// TwinCAT 3 PLC project PLC_DemoXTS
// ProgramVersion: 3.1.4026.17
// libraries:
//   Tc2_MC2, * (Beckhoff Automation GmbH)
//   Tc2_MC2_Camming, * (Beckhoff Automation GmbH)
//   Tc2_Standard, * (Beckhoff Automation GmbH)
//   Tc2_System, * (Beckhoff Automation GmbH)
//   Tc3_Mc3Definitions, * (Beckhoff Automation GmbH)
//   Tc3_McCollisionAvoidance, * (Beckhoff Automation GmbH)
//   Tc3_McCoordinatedMotion, * (Beckhoff Automation GmbH)
//   Tc3_Module, * (Beckhoff Automation GmbH)
// project tree:
//   GVLs/ GVL_Constant.TcGVL, GVL_XTS1.TcGVL, GVL_Infeed.TcGVL
//   / PlcTask.TcTTO
//   POUs/Infeed/ FB_Infeed.TcPOU, FB_VirtualMaster.TcPOU, Prg_Camming.TcPOU
//   POUs/ MAIN.TcPOU, XTS_MAIN.TcPOU
//   POUs/XTS/ FB_MoverCheckPos.TcPOU, FB_MoverCycle.TcPOU, FB_XTS.TcPOU, FB_AllMoversToStartpos.TcPOU
//   POUs/_NEW/Mover/ FB_MoverX.TcPOU, IMover.TcIO, ST_MoverData.TcDUT
//   POUs/_NEW/Position/ FB_PositionX.TcPOU, IPosition.TcIO
//   POUs/_NEW/Station/ FB_StationX.TcPOU, IStation.TcIO
//   POUs/_NEW/TrackList/ FB_Track.TcPOU, ITrack.TcIO

CONFIGURATION PLC_DemoXTS
    RESOURCE PLC ON TwinCAT3
        TASK PlcTask(INTERVAL := T#10ms, PRIORITY := 20);
        PROGRAM MAIN WITH PlcTask : MAIN;
    END_RESOURCE
END_CONFIGURATION

// ---- POUs/_NEW/Mover/ST_MoverData.TcDUT
TYPE ST_MoverData :
STRUCT
	id : UDINT;
	pos : LREAL;
	status : INT;
	assigned : BOOL;
END_STRUCT
END_TYPE

// ---- GVLs/GVL_Constant.TcGVL
VAR_GLOBAL CONSTANT
	iMaxNumbMovers		: INT := 35;
	iMaxNumbVirtMasters	: INT := 5;
END_VAR

// ---- GVLs/GVL_XTS1.TcGVL
{attribute 'qualified_only'}
VAR_GLOBAL CONSTANT
	
	iNumbOfMovers		: INT	:= 35;
	rRailLength			: LREAL	:= 6000.0;

END_VAR


VAR_GLOBAL

	Mover				: ARRAY [1..iNumbOfMovers] OF Axis_Ref;
	CAGroup				: AXES_GROUP_REF;		

	rInitPosition		: LREAL := 1100;
	rInitVelocity		: LREAL	:= 720;
	rGap				: LREAL	:= 90;
	rMasterVelocity		: LREAL	:= 600;
	rSlaveSyncPos		: LREAL := 1300;
	rSyncDistance		: LREAL := 400;
	rXTS_Velocity		: LREAL := 720;
	rRobot1_Position	: LREAL := 4000;
	rRobot2_Position	: LREAL := 5500;
	tTime_Robot1		: TIME := T#4500MS;
	tTime_Robot2		: TIME := T#1500MS;
	
END_VAR

// ---- GVLs/GVL_Infeed.TcGVL
{attribute 'qualified_only'}
VAR_GLOBAL CONSTANT
	
	iNumbOfVirtMasters		: INT	:= 4;

END_VAR


VAR_GLOBAL

	MasterAxis				: AXIS_REF;
	VirtalMaster			: ARRAY [1..iNumbOfVirtMasters] OF Axis_Ref;

	iProductsPerMinute		: INT 	:= 60;

	rDiameterWheel			: LREAL := 480;			// Diameter Infeed Wheel
	rMasterDistance_1Cycle	: LREAL := 360;			// 8 cycles per rotation
	rSyncPosition_Wheel_XTS	: LREAL := 471.5;		
	rDetectionPosMin		: LREAL := 160;
	rDetectionPosMax		: LREAL := 200;
	
	//CamTable
	rMasterDistance_P2		: LREAL	:= 180;
	rSlaveOffset_P2			: LREAL := 0;
	rMasterDistance_P3		: LREAL	:= 20;
	rSlaveOffset_P3			: LREAL	:= 10;
	rMasterDistance_P5		: LREAL := 30;
	rSlaveOffset_P5			: LREAL;
	rMasterDistance_P6		: LREAL := 180;
	rSlaveOffset_P6			: LREAL := -5;
	rSlaveOffset			: LREAL;
	
END_VAR

// ---- POUs/_NEW/Mover/IMover.TcIO
INTERFACE IMover

METHOD AssignAxisRef : bool
VAR_INPUT
	axis : REFERENCE TO AXIS_REF;
END_VAR
END_METHOD

METHOD AssignID : bool
VAR_INPUT
	ID : UDINT;
END_VAR
END_METHOD

METHOD GetPosition : LREAL
VAR_INPUT
END_VAR
END_METHOD

METHOD GetStatus : int
VAR_INPUT
END_VAR
END_METHOD

METHOD SetPositionID : BOOL
VAR_INPUT
	ID: UDINT;
END_VAR
END_METHOD

METHOD SetStatus : BOOL;
VAR_INPUT
	status : INT;
END_VAR
END_METHOD

METHOD UpdateData : ST_MoverData
VAR_INPUT
END_VAR
END_METHOD

METHOD UpdatePosition : bool
VAR_INPUT
END_VAR
END_METHOD

END_INTERFACE

// ---- POUs/_NEW/Position/IPosition.TcIO
INTERFACE IPosition

METHOD Available : bool
VAR_INPUT
END_VAR
END_METHOD

METHOD Disable : BOOL
VAR_INPUT
END_VAR
END_METHOD

METHOD Enable : BOOL
VAR_INPUT
END_VAR
END_METHOD

METHOD GetID : UDINT
VAR_INPUT
END_VAR
END_METHOD

METHOD GetPosition : LREAL
VAR_INPUT
END_VAR
END_METHOD

METHOD SetID : BOOL
VAR_INPUT
	ID : UDINT;
END_VAR
END_METHOD

METHOD SetMover : bool
VAR_INPUT
	moverNumber : UDINT;
END_VAR
END_METHOD

METHOD SetPosition
VAR_INPUT
	position : LREAL;
END_VAR
END_METHOD

END_INTERFACE

// ---- POUs/_NEW/Station/IStation.TcIO
INTERFACE IStation

METHOD FindMoverMatch : udint
VAR_INPUT
END_VAR
END_METHOD

METHOD FindNextPosition : IPosition;
VAR_INPUT
END_VAR
END_METHOD

METHOD GetMovers : BOOL
VAR_INPUT
END_VAR
END_METHOD

METHOD SetPosRef : BOOL
VAR_INPUT
	PosIndex : DINT;
	PosRef	: REFERENCE TO FB_PositionX;
END_VAR
END_METHOD

METHOD SetStationAttraction : BOOL
VAR_INPUT
	setState : INT;
END_VAR
END_METHOD

METHOD SetTrackRef : BOOL
VAR_INPUT
	TrackRef : ITrack;
END_VAR
END_METHOD

END_INTERFACE

// ---- POUs/_NEW/TrackList/ITrack.TcIO
INTERFACE ITrack

METHOD FindMover : UDINT
VAR_INPUT
	status : INT;
END_VAR
END_METHOD

METHOD SetMoverInUse : BOOL;
VAR_INPUT
	moverNumber	: UDINT;
END_VAR
END_METHOD

METHOD SetMoverRef : BOOL
VAR_INPUT
	index : DINT;
	mover	: IMover;
END_VAR
END_METHOD

METHOD Sort : bool
VAR_INPUT
END_VAR
END_METHOD

METHOD UpdateMoverData : bool
VAR_INPUT
	data	: ST_MoverData;
END_VAR
END_METHOD

END_INTERFACE

// ---- POUs/MAIN.TcPOU
PROGRAM MAIN
VAR

	bEnable_XTS1			: BOOL;
	bMoveToStartPos_XTS1	: BOOL;
	bEnable_Master			: BOOL;
	bMoveMaster				: BOOL;
	bSensor_Product			: BOOL;

	fbInfeed1				: FB_Infeed;
	fbXTS1					: FB_XTS;
	fbMoveToStartPos_XTS1	: FB_AllMoversToStartpos;
	
	// Cycle
	i,j						: INT;
	bStartSyncMaster		: BOOL;
	bStartSyncMover			: BOOL;
	Trg_bStartSyncMaster	: R_Trig;
	iMoverAtStartpos_XTS1	: INT;
	iVirtMasterAtStartpos	: INT;
	fbMoveratStartPos_XTS1	: ARRAY [1..GVL_XTS1.iNumbOfMovers] OF FB_MoverCheckPos;
	fbMoveratRobot1Pos		: ARRAY [1..GVL_XTS1.iNumbOfMovers] OF FB_MoverCheckPos;
	fbMoveratRobot2Pos		: ARRAY [1..GVL_XTS1.iNumbOfMovers] OF FB_MoverCheckPos;
	fbMoverCycle_XTS1		: ARRAY [1..GVL_XTS1.iNumbOfMovers] OF FB_MoverCycle;
	
	// Robot1 and Robot2
	MoverAtRobot1			: ARRAY [1..10] OF INT;
	MoverAtRobot2			: ARRAY [1..10] OF INT;
	bRobot1_Filled			: BOOL;
	bRobot2_Filled			: BOOL;
	fbRobot1_Timer			: TON;
	fbRobot2_Timer			: TON;
	
	MyXTS	: XTS_MAIN;

END_VAR

Prg_Camming();

// Infeed
fbInfeed1(
	bEnable_Master		:= bEnable_Master, 
	bMoveMaster			:= bMoveMaster, 
	bSensorProduct		:= bSensor_Product,
	Master				:= GVL_Infeed.MasterAxis, 
	VirtMaster			:= GVL_Infeed.VirtalMaster,
	);


// XTS 1 : Enable all movers with Collision Avoindance
fbXTS1(
	bEnable_XTS		:= bEnable_XTS1, 
	Mover			:= GVL_XTS1.Mover, 
	CAGroup			:= GVL_XTS1.CAGroup, 
	);
	
	
// XTS 1 : Move all movers to Startposition 
fbMoveToStartPos_XTS1(
	bXTS_MoveToStartPos	:= bMoveToStartPos_XTS1, 
	rInitPosition		:= GVL_XTS1.rInitPosition, 
	rInitVelocity		:= GVL_XTS1.rInitVelocity, 
	rRailLength			:= GVL_XTS1.rRailLength, 
	rGap				:= GVL_XTS1.rGap, 
	Mover				:= GVL_XTS1.Mover,
	);

	
// XTS 1 : Find which mover is waiting at Startposition	
iMoverAtStartpos_XTS1 := 0;
FOR i:=1 TO GVL_XTS1.iNumbOfMovers DO
	fbMoveratStartPos_XTS1[i](
		rActualPosition	:= GVL_XTS1.Mover[i].NcToPlc.ModuloSetPos, 
		rCheckPosition	:= GVL_XTS1.rInitPosition, 
		rRailLength		:= GVL_XTS1.rRailLength
		);
	IF fbMoveratStartPos_XTS1[i].bInPosition THEN
		iMoverAtStartpos_XTS1 := i;
	END_IF
	
END_FOR
	
// Start Synchronisation Virtual Master
bStartSyncMaster:=FALSE;
iVirtMasterAtStartpos:=0;
FOR i := 1 TO GVL_Infeed.iNumbOfVirtMasters DO
	IF (GVL_Infeed.VirtalMaster[i].NcToPlc.SetPos>GVL_Infeed.rSlaveOffset+10) AND (GVL_Infeed.VirtalMaster[i].NcToPlc.SetPos<GVL_Infeed.rSlaveOffset+120) THEN
		iVirtMasterAtStartpos:=i;
		bStartSyncMaster:=TRUE;
	END_IF
END_FOR

// Start Synchronisation Mover
Trg_bStartSyncMaster(Clk:=bStartSyncMaster);
IF (iMoverAtStartpos_XTS1<>0) AND Trg_bStartSyncMaster.Q THEN
	bStartSyncMover:=TRUE;
END_IF
IF iMoverAtStartpos_XTS1=0 OR NOT bStartSyncMaster THEN
	bStartSyncMover:=FALSE;
END_IF

// XTS 1 : Cyclic movement for all movers
FOR i:=1 TO GVL_XTS1.iNumbOfMovers DO
	fbMoverCycle_XTS1[i](
		bStartCycle			:= bStartSyncMover AND (iMoverAtStartpos_XTS1=i), 
		iVirtMasterAtStart	:= iVirtMasterAtStartpos,
		rMasterSyncPos		:= 300,
		rSlaveSyncPos		:= (GVL_XTS1.Mover[i].NcToPlc.ModuloActTurns * GVL_XTS1.rRailLength) + GVL_XTS1.rSlaveSyncPos,
		Mover				:= GVL_XTS1.Mover[i]
		);

END_FOR

// Cyclus Pers + Robot1 

FOR j := 1 TO 10 DO
	MoverAtRobot1[j] := 0;
	FOR i:=1 TO GVL_XTS1.iNumbOfMovers DO
		fbMoveratRobot1Pos[i](
			rActualPosition	:= GVL_XTS1.Mover[i].NcToPlc.ModuloSetPos, 
			rCheckPosition	:= GVL_XTS1.rRobot1_Position - (j*GVL_XTS1.rGap) + GVL_XTS1.rGap , 
			rRailLength		:= GVL_XTS1.rRailLength
			);
		IF fbMoveratRobot1Pos[i].bInPosition THEN
			MoverAtRobot1[j] := i;
		END_IF
	END_FOR
END_FOR

bRobot1_Filled := TRUE;
FOR i := 1 TO 10 DO
	IF MoverAtRobot1[i]=0 THEN
		bRobot1_Filled := FALSE;
	END_IF
END_FOR

fbRobot1_Timer(IN:=bRobot1_Filled , PT:=GVL_XTS1.tTime_Robot1 );
IF fbRobot1_Timer.Q THEN
	FOR i:=1 TO 10 DO
		fbMoverCycle_XTS1[MoverAtRobot1[i]].Robot1_Ready:=TRUE;	
	END_FOR
ELSE
	FOR i:=1 TO GVL_XTS1.iNumbOfMovers DO
		fbMoverCycle_XTS1[i].Robot1_Ready:=FALSE;	
	END_FOR	
END_IF


// Cyclus Robot2 

FOR j := 1 TO 10 DO
	MoverAtRobot2[j] := 0;
	FOR i:=1 TO GVL_XTS1.iNumbOfMovers DO
		fbMoveratRobot2Pos[i](
			rActualPosition	:= GVL_XTS1.Mover[i].NcToPlc.ModuloSetPos, 
			rCheckPosition	:= GVL_XTS1.rRobot2_Position - (j*GVL_XTS1.rGap) + GVL_XTS1.rGap , 
			rRailLength		:= GVL_XTS1.rRailLength
			);
		IF fbMoveratRobot2Pos[i].bInPosition THEN
			MoverAtRobot2[j] := i;
		END_IF
	END_FOR
END_FOR

bRobot2_Filled := TRUE;
FOR i := 1 TO 10 DO
	IF MoverAtRobot2[i]=0 THEN
		bRobot2_Filled := FALSE;
	END_IF
END_FOR

fbRobot2_Timer(IN:=bRobot2_Filled , PT:=GVL_XTS1.tTime_Robot2 );
IF fbRobot2_Timer.Q THEN
	FOR i:=1 TO 10 DO
		fbMoverCycle_XTS1[MoverAtRobot2[i]].Robot2_Ready:=TRUE;	
	END_FOR
ELSE
	FOR i:=1 TO GVL_XTS1.iNumbOfMovers DO
		fbMoverCycle_XTS1[i].Robot2_Ready:=FALSE;	
	END_FOR	
END_IF

// call
MyXTS(axisRef := GVL_XTS1.Mover);

END_PROGRAM

// ---- POUs/Infeed/FB_Infeed.TcPOU
FUNCTION_BLOCK FB_Infeed
VAR_INPUT
	bEnable_Master			: BOOL;
	bMoveMaster				: BOOL;
	bSensorProduct			: BOOL;
END_VAR

VAR_IN_OUT
	Master					: Axis_Ref;
	VirtMaster				: ARRAY [*] OF Axis_Ref;
END_VAR

VAR
	i						: DINT;
	iStartIndex				: DINT;
	VeloMaster				: LREAL;
	bToggle					: BOOL;

	fbPowerMaster			: MC_Power;
	fbMoveMaster			: MC_MoveVelocity;
	fbStopMaster			: MC_Halt;
	fbPowerVirtMaster		: ARRAY [1..iMaxNumbVirtMasters] OF MC_Power;
	fbVirtMaster			: ARRAY [1..iMaxNumbVirtMasters] OF FB_VirtualMaster;

END_VAR

// Enable Master
Master.ReadStatus();
fbPowerMaster(
	Axis			:= Master, 
	Enable			:= bEnable_Master, 
	Enable_Positive	:= bEnable_Master, 
	Enable_Negative	:= bEnable_Master, 
	Override		:= 100, 
	);
	
FOR i := 1 TO UPPER_BOUND(VirtMaster,1) DO
	VirtMaster[i].ReadStatus();
	fbPowerVirtMaster[i](
		Axis			:= VirtMaster[i], 
		Enable			:= bEnable_Master, 
		Enable_Positive	:= bEnable_Master, 
		Enable_Negative	:= bEnable_Master, 
		Override		:= 100, 
		);
END_FOR


// Start-Stop Master

VeloMaster := GVL_Infeed.iProductsPerMinute * 360 / 60;
bToggle:=NOT bToggle;

fbMoveMaster(
	Axis		:= Master, 
	Execute		:= bMoveMaster AND bToggle, 
	Velocity	:= VeloMaster, 
	Direction	:= MC_Positive_Direction, 
	);
fbStopMaster(
	Axis		:= Master, 
	Execute		:= NOT bMoveMaster, 
	);

// Virtual Master ready to start
iStartIndex:=0;
FOR i := 1 TO UPPER_BOUND(VirtMaster,1) DO
	IF VirtMaster[i].NcToPlc.ActPos=0 THEN
		iStartIndex:=i;
		i:=5;
	END_IF
END_FOR
	
// Detection product
FOR i := 1 TO UPPER_BOUND(VirtMaster,1) DO
	fbVirtMaster[i].bActivateCam:=FALSE;
END_FOR

IF (Master.NcToPlc.ModuloActPos > GVL_Infeed.rDetectionPosMin) AND (Master.NcToPlc.ModuloActPos < GVL_Infeed.rDetectionPosMax) AND bSensorProduct THEN
	fbVirtMaster[iStartIndex].bActivateCam:=TRUE;
END_IF
 
FOR i := 1 TO UPPER_BOUND(VirtMaster,1) DO
	fbVirtMaster[i](
		Master:= Master, 
		Slave:= VirtMaster[i],
		);
END_FOR

END_FUNCTION_BLOCK

// ---- POUs/Infeed/FB_VirtualMaster.TcPOU
FUNCTION_BLOCK FB_VirtualMaster
VAR_INPUT
	bActivateCam	: BOOL;
END_VAR
VAR_OUTPUT
END_VAR
VAR_IN_OUT
	Master			: Axis_Ref;
	Slave			: Axis_Ref;
END_VAR
VAR
	fbCamIn			: MC_CamIn;
	Options			: ST_CamInOptions;
	fbCamOut		: MC_CamOut;
	fbStop			: MC_Halt;
	fbSetPos		: MC_SetPosition;
	MasterOffset	: LREAL;;
END_VAR

Options.ActivationMode := MC_CamActivationMode.MC_CAMACTIVATION_ATMASTERAXISPOS;
Options.ActivationPosition := (Master.NcToPlc.ModuloActTurns+1)*360;
CASE (Master.NcToPlc.ModuloActTurns MOD 3) OF
0:	MasterOffset:=720;
1:	MasterOffset:=360;
2:	MasterOffset:=0;
END_CASE


fbCamIn(
	Master			:= Master, 
	Slave			:= Slave, 
	Execute			:= bActivateCam, 
	StartMode		:= MC_StartMode.MC_STARTMODE_MASTERABS_SLAVEREL,
	MasterOffset	:= MasterOffset,
	CamTableID		:= 1, 
	Options			:= Options, 
	);

fbCamOut.Execute	:= FALSE;
fbStop.Execute 		:= FALSE;
fbSetPos.Execute 	:= FALSE;
IF Slave.NcToPlc.ActPos>750 THEN
	fbCamOut.Execute := TRUE;
	IF fbCamOut.Done THEN fbStop.Execute := TRUE; END_IF
	IF fbStop.Done THEN fbSetPos.Execute := TRUE; END_IF
END_IF

fbCamOut	(Slave	:= Slave);	
fbStop		(Axis	:= Slave);
fbSetPos	(Axis	:= Slave);

END_FUNCTION_BLOCK

// ---- POUs/XTS/FB_XTS.TcPOU
FUNCTION_BLOCK FB_XTS

VAR_INPUT
	bEnable_XTS				: BOOL;
END_VAR

VAR_IN_OUT
	Mover					: ARRAY [*] OF AXIS_REF;
	CAGroup					: AXES_GROUP_REF;
END_VAR

VAR_OUTPUT
	// Status bits	
	bAllMoversFound			: BOOL;
	bAllMoversEnabled		: BOOL;
	bMoverHasError			: BOOL;
	bCAGroupMoving			: BOOL;
	bCAGroupError			: BOOL;
	bCAGroupNotReady		: BOOL;
	bCAGroupStandby			: BOOL;
	bCAGroupStopping		: BOOL;
	bCAGroupDisabled		: BOOL;
END_VAR

VAR
	i						: DINT;
	step					: INT;
	pMover					: POINTER TO AXIS_REF;

	// Command bits
	bResetAll				: BOOL;
	bEnableAllMovers		: BOOL;
	bEnableCAGroup			: BOOL;
	bDisableCAGroup			: BOOL;
	bResetMovers			: BOOL;
	bResetCAGroup			: BOOL;
	bConfig_CAGroup			: BOOL;
	bReConfig_CAGroup		: BOOL;

	// Status bits	
	bRunXTS					: BOOL;
	bConfig_CAGroupDone		: BOOL;
	bConfig_CAGroupErr		: BOOL;
	bReConfig_CAGroupDone	: BOOL;
	bReConfig_CAGroupErr	: BOOL;

	// Function Blocks
	fbPowerMover			: ARRAY [1..iMaxNumbMovers] OF MC_Power;
	fbResetMover			: ARRAY [1..iMaxNumbMovers] OF MC_Reset;
	fbAddAxisTo_CAGroup		: ARRAY [1..iMaxNumbMovers] OF MC_AddAxisToGroup;
	fbRemoveFrom_CAGroup	: ARRAY [1..iMaxNumbMovers] OF MC_RemoveAxisFromGroup;
	fbEnableCAGroup			: MC_GroupEnable;
	fbDisableCAGroup		: MC_GroupDisable;
	fbResetCAGroup			: MC_GroupReset;
	fbCAGroupReadStatus		: MC_GroupReadStatus;
	fbTimer					: TON;
	fbRTrgReset				: R_TRIG;	
END_VAR


// **************************************************************************************
// Wait until XTS is started
// **************************************************************************************

IF NOT bRunXTS THEN
	bAllMoversFound := TRUE;
	FOR i:=1 TO UPPER_BOUND(Mover,1) DO
		bAllMoversFound := bAllMoversFound AND Mover[i].NcToPlc.ActPos<>0;
	END_FOR
	bRunXTS := bAllMoversFound;
END_IF

IF NOT bRunXTS THEN
	RETURN;
END_IF


// **************************************************************************************
// Init XTS with Collision Avoidance
// **************************************************************************************

CASE step OF
	
0:		// Wait for Enable-XTS command
		bResetCAGroup 			:= fbRTrgReset.Q;
		bResetMovers			:= fbRTrgReset.Q;	 
		bEnableCAGroup			:= FALSE;
		bDisableCAGroup			:= FALSE;
		bConfig_CAGroupDone		:= FALSE;
		bConfig_CAGroupErr		:= FALSE;
		bReConfig_CAGroupDone	:= FALSE;
		bReConfig_CAGroupErr	:= FALSE;
		IF bEnable_XTS THEN
			Step:=10;	
		END_IF
	
10:		//Add Axis to Group
		bConfig_CAGroup:=TRUE;
		IF bConfig_CAGroupDone THEN
			Step:=20;
			bConfig_CAGroup:=FALSE;
		END_IF
		IF bConfig_CAGroupErr THEN
			Step:=999;
			bConfig_CAGroup:=FALSE;
		END_IF
		
20:		//Enable CA-Group
		bEnableCAGroup:=TRUE;
		IF fbEnableCAGroup.Done THEN
			Step:=30;
			bEnableCAGroup:=FALSE;
		END_IF
		IF fbEnableCAGroup.Error THEN
			Step:=999;
			bEnableCAGroup:=FALSE;
		END_IF	
		
30:		// Power Movers
		bEnableAllMovers := TRUE;
		fbTimer(IN:=TRUE,PT:=T#200MS);
		IF fbTimer.Q THEN
			Step:=40;
			fbTimer(IN:=FALSE);
		END_IF
			
40:		// Reset Movers
		bResetMovers := TRUE;
		fbTimer(IN:=TRUE,PT:=T#2000MS);
		IF bAllMoversEnabled THEN
			Step:=50;
			bResetMovers := FALSE;
			fbTimer(IN:=FALSE);
		END_IF
		IF fbTimer.Q THEN 
			Step:=999;
			bResetMovers := FALSE;
			fbTimer(IN:=FALSE);
		END_IF
	
50:		// Reset CA-Group
		bResetCAGroup := TRUE;
		IF fbResetCAGroup.Done THEN
			Step:=100;
			bResetCAGroup := FALSE;
		END_IF
		IF fbResetCAGroup.Error THEN
			Step:=999;
			bResetCAGroup := FALSE;
		END_IF	
	
100:	// XTS CA-Group Ready
		bResetCAGroup 	:= fbRTrgReset.Q;
		bResetMovers	:= fbRTrgReset.Q;	 
		IF NOT bEnable_XTS THEN
			Step:=110;
		END_IF

110:	// Disable Movers
		bEnableAllMovers := FALSE;
		fbTimer(IN:=TRUE,PT:=T#200MS);
		IF fbTimer.Q THEN
			Step:=120;
			fbTimer(IN:=FALSE);
		END_IF
	
120:	// Disable CA-Group		
		bDisableCAGroup:=TRUE;
		IF fbDisableCAGroup.Done THEN
			Step:=130;
			bDisableCAGroup:=FALSE;
			bEnableAllMovers:=FALSE;
		END_IF
		IF fbDisableCAGroup.Error THEN
			Step:=999;
			bDisableCAGroup:=FALSE;
		END_IF		

130:	// Reconfig CA-Group
		bReConfig_CAGroup:=TRUE;
		IF bReConfig_CAGroupDone THEN
			Step:=140;
			bReConfig_CAGroup:=FALSE;
		END_IF
		IF bReConfig_CAGroupErr THEN
			Step:=999;
			bReConfig_CAGroup:=FALSE;
		END_IF
		M_Config_CAGroup();
		
140:	// Reset Movers
		bResetMovers := TRUE;
		fbTimer(IN:=TRUE,PT:=T#2000MS);
		IF NOT bMoverHasError THEN
			Step:=150;
			bResetMovers := FALSE;
			fbTimer(IN:=FALSE);
		END_IF
		IF fbTimer.Q THEN 
			Step:=999;
			bResetMovers := FALSE;
			fbTimer(IN:=FALSE);
		END_IF

150:	// Reset CA-Group
		bResetCAGroup := TRUE;
		IF fbResetCAGroup.Done THEN
			Step:=0;
			bResetCAGroup := FALSE;
		END_IF
		IF fbResetCAGroup.Error THEN
			Step:=999;
			bResetCAGroup := FALSE;
		END_IF	

999:	// Error
		bEnable_XTS			:=FALSE;
		bEnableAllMovers	:=FALSE;
		bResetCAGroup 		:= fbRTrgReset.Q;
		bResetMovers		:= fbRTrgReset.Q;	 
		IF fbRTrgReset.Q THEN
			Step:=0;
		END_IF

END_CASE

M_Config_CAGroup();
M_ReadStatus();
M_Enable_Movers();
M_Enable_CAGroup();
M_Reset();	

fbRTrgReset(CLK:=bResetAll);

METHOD M_Config_CAGroup 	: BOOL
VAR
END_VAR
// Add Axis to Group
FOR i := 1 TO UPPER_BOUND(Mover,1) DO
	bConfig_CAGroupDone	:= TRUE;
	fbAddAxisTo_CAGroup[i](
		AxesGroup		:= CAGroup, 
		Axis			:= Mover[i], 
		Execute			:= bConfig_CAGroup, 
		IdentInGroup	:= UDINT_TO_IDENTINGROUP(i), 
		);		
	bConfig_CAGroupDone	:= bConfig_CAGroupDone AND fbAddAxisTo_CAGroup[i].Done;
	bConfig_CAGroupErr	:= bConfig_CAGroupErr OR fbAddAxisTo_CAGroup[i].Error;
END_FOR

// Remove Axis from Group
FOR i := 1 TO UPPER_BOUND(Mover,1) DO
	bReConfig_CAGroupDone	:= TRUE;
	fbRemoveFrom_CAGroup[i](
		AxesGroup			:= CAGroup, 
		Execute				:= bReConfig_CAGroup, 
		IdentInGroup		:= UDINT_TO_IDENTINGROUP(i), 
		);
	bReConfig_CAGroupDone	:= bReConfig_CAGroupDone AND fbRemoveFrom_CAGroup[i].Done;
	bReConfig_CAGroupErr	:= bReConfig_CAGroupErr OR fbRemoveFrom_CAGroup[i].Error;
END_FOR
END_METHOD

METHOD M_Enable_CAGroup : BOOL
VAR_INPUT
END_VAR
// Enable CA-Group
fbEnableCAGroup(
	AxesGroup	:= CAGroup, 
	Execute		:= bEnableCAGroup, 
	);	

	
// Disable CA-Group	
fbDisableCAGroup(
	AxesGroup	:= CAGroup, 
	Execute		:= bDisableCAGroup, 
	);
END_METHOD

METHOD M_Enable_Movers : BOOL
VAR_INPUT
END_VAR
// Enable Movers
FOR i:=1 TO UPPER_BOUND(Mover,1) DO
	fbPowerMover[i](
		Axis			:= Mover[i], 
		Enable			:= bEnableAllMovers, 
		Enable_Positive	:= bEnableAllMovers, 
		Enable_Negative	:= bEnableAllMovers, 
		Override		:= 100, 
		);
END_FOR
END_METHOD

METHOD M_ReadStatus : BOOL
VAR_INPUT
END_VAR
// All Movers Enabled
bAllMoversEnabled := TRUE;
FOR i:=1 TO UPPER_BOUND(Mover,1) DO
	bAllMoversEnabled := bAllMoversEnabled AND Mover[i].Status.ControlLoopClosed;
END_FOR

// Mover has Error
bMoverHasError := FALSE;
FOR i:=1 TO UPPER_BOUND(Mover,1) DO
	bMoverHasError := bMoverHasError OR Mover[i].Status.Error;
END_FOR

// Read Status NC
FOR i:=1 TO UPPER_BOUND(Mover,1) DO
	Mover[i].ReadStatus();
END_FOR

// Read Status CA-Group
fbCAGroupReadStatus(
	AxesGroup		:= CAGroup, 
	Enable			:= NOT fbCAGroupReadStatus.Busy, 
	GroupMoving		=> bCAGroupMoving, 
	GroupErrorStop	=> bCAGroupError, 
	GroupNotReady	=> bCAGroupNotReady, 
	GroupStandby	=> bCAGroupStandby, 
	GroupStopping	=> bCAGroupStopping, 
	GroupDisabled	=> bCAGroupDisabled, 
	);
END_METHOD

METHOD M_Reset : BOOL
VAR_INPUT
END_VAR
// Reset Movers
FOR i:=1 TO UPPER_BOUND(Mover,1) DO
	fbResetMover[i](
		Axis	:= Mover[i], 
		Execute	:= bResetMovers (*AND Mover[i].Status.Error*) 
		);
END_FOR

// Reset CA-Group
fbResetCAGroup(
	AxesGroup	:= CAGroup, 
	Execute		:= bResetCAGroup, 
	);
END_METHOD

END_FUNCTION_BLOCK

// ---- POUs/XTS/FB_AllMoversToStartpos.TcPOU
FUNCTION_BLOCK FB_AllMoversToStartpos
VAR_INPUT
	bXTS_MoveToStartPos		: BOOL;
	rInitPosition			: LREAL;
	rInitVelocity			: LREAL;
	rRailLength				: LREAL;
	rGap					: LREAL;
END_VAR

VAR_IN_OUT
	Mover					: ARRAY [*] OF AXIS_REF;
END_VAR

VAR
	i						: DINT;
	fbMoveToStartPos		: ARRAY [1..iMaxNumbMovers] OF MC_MoveRelativeCA;
END_VAR

// **************************************************************************************
// Move all Movers to initial position
// **************************************************************************************

FOR i:=1 TO UPPER_BOUND(Mover,1) DO
	
	IF Mover[i].NcToPlc.ModuloSetPos < (rInitPosition - 1) THEN
		fbMoveToStartPos[i].Distance := rInitPosition - Mover[i].NcToPlc.ModuloSetPos;
	ELSE;
		fbMoveToStartPos[i].Distance := rInitPosition - Mover[i].NcToPlc.ModuloSetPos + rRailLength ;
	END_IF
		
	fbMoveToStartPos[i](
		Axis			:= Mover[i], 
		Execute			:= bXTS_MoveToStartPos, 
		ContinuousUpdate:= TRUE, 
		Velocity		:= rInitVelocity, 
		Gap				:= rGap, 
		);

END_FOR

END_FUNCTION_BLOCK

// ---- POUs/XTS/FB_MoverCheckPos.TcPOU
FUNCTION_BLOCK FB_MoverCheckPos
VAR_INPUT
	rActualPosition	: LREAL;
	rCheckPosition	: LREAL;
	rRailLength		: LREAL;
END_VAR
VAR_OUTPUT
	bInPosition		: BOOL;
END_VAR
VAR
	rTolerance		: LREAL	:= 1;
END_VAR

bInPosition:=FALSE;
IF rCheckPosition<=rTolerance THEN
	IF rActualPosition>(rRailLength+rCheckPosition-rTolerance) OR rActualPosition<(rCheckPosition+rTolerance) THEN
		bInPosition:=TRUE;
	END_IF
END_IF

IF rCheckPosition>rTolerance AND rCheckPosition<(rRailLength-rTolerance) THEN
	IF rActualPosition>(rCheckPosition-rTolerance) AND rActualPosition<(rCheckPosition+rTolerance)THEN
		bInPosition:=TRUE;
	END_IF
END_IF

IF rCheckPosition>=(rRailLength-rTolerance) THEN
	IF rActualPosition>(rCheckPosition-rTolerance) OR rActualPosition<(rCheckPosition+rTolerance-rRailLength)THEN
		bInPosition:=TRUE;
	END_IF
END_IF

END_FUNCTION_BLOCK

// ---- POUs/XTS/FB_MoverCycle.TcPOU
FUNCTION_BLOCK FB_MoverCycle 
VAR_INPUT
	bStartCycle			: BOOL;
	iVirtMasterAtStart	: int;
	rMasterSyncPos		: MC_LREAL;
	rSlaveSyncPos		: MC_LREAL;
	Robot1_Ready		: BOOL;
	Robot2_Ready		: BOOL;
END_VAR
VAR_OUTPUT
END_VAR
VAR_IN_OUT
	Mover				: AXIS_REF;
END_VAR
VAR
	i					: INT;
	step				: INT;
	fbGearIn			: MC_GearInPosCA;
	fbMoveToRobot1		: MC_MoveAbsoluteCA;
	fbMoveToRobot2		: MC_MoveAbsoluteCA;
	fbMoveStartPos		: MC_MoveAbsoluteCA;
END_VAR

CASE step OF
	
	0:	// Wait for startcommand
	
		fbGearIn.Execute		:= FALSE;	
		fbMoveStartPos.Execute 	:= FALSE;
		fbMoveToRobot1.Execute	:= FALSE;	
		fbMoveToRobot2.Execute	:= FALSE;	
	
		IF bStartCycle THEN
			step:=10;
		END_IF
		
	
	10:	// Sync with Master

		fbGearIn.Execute				:= TRUE; 
		fbGearIn.ContinuousUpdate		:= TRUE; 
		fbGearIn.RatioNumerator			:= 1; 
		fbGearIn.RatioDenumerator		:= 1; 
		fbGearIn.MasterSyncPosition		:= rMasterSyncPos; 
		fbGearIn.SlaveSyncPosition		:= rSlaveSyncPos; 
		fbGearIn.SyncStrategy			:= mcSyncStrategyEarly; 
		fbGearIn.Velocity				:= 4000;

		IF Mover.NcToPlc.ModuloActPos > (GVL_XTS1.rSlaveSyncPos+GVL_XTS1.rSyncDistance) THEN
			step:=20;
		END_IF

	20:	// Move To Robot1	
		
		fbMoveToRobot1.Position			:= (Mover.NcToPlc.ModuloActTurns * GVL_XTS1.rRailLength) + GVL_XTS1.rRobot1_Position;
		fbMoveToRobot1.Velocity 		:= GVL_XTS1.rXTS_Velocity;
		fbMoveToRobot1.ContinuousUpdate	:= FALSE;
		fbMoveToRobot1.Gap				:= GVL_XTS1.rGap;
		fbMoveToRobot1.BufferMode		:= mcAborting;
		fbMoveToRobot1.Execute			:= TRUE;
		
		IF Robot1_Ready THEN
			step:=30;
		END_IF
		
	30:	// Move To Robot2	
		
		fbMoveToRobot2.Position			:= (Mover.NcToPlc.ModuloActTurns * GVL_XTS1.rRailLength) + GVL_XTS1.rRobot2_Position;
		fbMoveToRobot2.Velocity 		:= GVL_XTS1.rXTS_Velocity;
		fbMoveToRobot2.ContinuousUpdate	:= FALSE;
		fbMoveToRobot2.Gap				:= GVL_XTS1.rGap;
		fbMoveToRobot2.BufferMode		:= mcAborting;
		fbMoveToRobot2.Execute			:= TRUE;
		
		IF Robot2_Ready THEN
			step:=40;
		END_IF
	
	40:	// Goto startposition

		fbMoveStartPos.Position			:= (Mover.NcToPlc.ModuloActTurns * GVL_XTS1.rRailLength) + GVL_XTS1.rInitPosition + GVL_XTS1.rRailLength;
		fbMoveStartPos.Velocity 		:= GVL_XTS1.rXTS_Velocity;
		fbMoveStartPos.ContinuousUpdate	:= FALSE;
		fbMoveStartPos.Gap				:= GVL_XTS1.rGap;
		fbMoveStartPos.BufferMode		:= mcAborting;
		fbMoveStartPos.Execute			:= TRUE;
		IF fbMoveStartPos.Done THEN
			step:=0;
		END_IF
		

END_CASE

fbMoveStartPos	( Axis:= Mover);
fbMoveToRobot1	( Axis:= Mover);
fbMoveToRobot2	( Axis:= Mover);
fbGearIn		( Master:= GVL_Infeed.VirtalMaster[iVirtMasterAtStart], Slave:= Mover);

END_FUNCTION_BLOCK

// ---- POUs/XTS_MAIN.TcPOU
FUNCTION_BLOCK XTS_MAIN
VAR_IN_OUT
	axisRef : ARRAY [1..iMaxNumbMovers] OF AXIS_REF;
END_VAR
VAR
	fbMover	: ARRAY [1..iMaxNumbMovers] OF FB_MoverX;
	fbPosition	: ARRAY [1..10] OF FB_PositionX;
	initDone : BOOL;
	i : DINT;
	positionActive : DINT;
	size : DINT;
	position : INT;
	list : ARRAY [1..iMaxNumbMovers] OF ST_MoverData;
	trackList : FB_Track;
	foundMover : UDINT;
	id : UDINT;
	IPosition : IPosition;
	IMover : IMover;
	statusRequest : INT := 1;
	station : FB_StationX;

END_VAR

// Init
IF NOT initDone THEN
	// Reference Axis to Mover Object
	FOR i:=1 TO iMaxNumbMovers DO
		fbMover[i].AssignID(ID:= i);
		fbMover[i].AssignAxisRef(axis:= axisRef[i]);
	END_FOR
	
	// Reference Movers to Track
	FOR i:=1 TO iMaxNumbMovers DO
		tracklist.SetMoverRef(
					index:= i, 
					mover:= fbMover[i]);
	END_FOR
	
	// Reference Positions to Stations
	FOR i:=1 TO 10 DO
	station.SetPosRef(
				PosIndex:= i, 
				PosRef:= fbPosition[i]);
	END_FOR
	
	// Reference Track to the Station
	station.SetTrackRef(trackList);
	
	// User Position Configuration
	FOR i:=1 TO 10 DO
		position := position + 100;
		fbPosition[i].SetPosition(position := position);
		fbPosition[i].SetID(LREAL_TO_UDINT(position));
	END_FOR
	initDone := TRUE;
END_IF


// Cyclic
FOR i:=1 TO iMaxNumbMovers DO
	trackList.UpdateMoverData(data := fbMover[i].UpdateData());
END_FOR
trackList.Sort();


station.GetMovers();

END_FUNCTION_BLOCK

// ---- POUs/_NEW/Mover/FB_MoverX.TcPOU
FUNCTION_BLOCK FB_MoverX IMPLEMENTS IMover
VAR
	_id       : UDINT;
	_axisRef  : REFERENCE TO AXIS_REF;
	_position : LREAL;
	_velocity : LREAL;
	_status	: INT;
	_posId	: UDINT;	
END_VAR

METHOD AssignAxisRef : BOOL
VAR_INPUT
	axis	: REFERENCE TO AXIS_REF;
END_VAR
_axisRef REF= axis;
AssignAxisRef := TRUE;
END_METHOD

METHOD AssignID : BOOL
VAR_INPUT
	ID	: UDINT;
END_VAR
_id := ID;
END_METHOD

METHOD GetPosition : LREAL
GetPosition := _position;
END_METHOD

METHOD GetStatus : INT
GetStatus := _status;
END_METHOD

METHOD SetPositionID : BOOL
VAR_INPUT
	ID	: UDINT;
END_VAR
_posId := ID;
END_METHOD

METHOD SetStatus : BOOL
VAR_INPUT
	status	: INT;
END_VAR
_status := status;
SetStatus := true;
END_METHOD

METHOD UpdateData : ST_MoverData
_position := _axisRef.NcToPlc.ModuloActPos;
UpdateData.id := _id;
UpdateData.pos := _position;
UpdateData.status := _status;
END_METHOD

METHOD UpdatePosition : BOOL
_position := _axisRef.NcToPlc.ModuloActPos;
END_METHOD

END_FUNCTION_BLOCK

// ---- POUs/_NEW/Position/FB_PositionX.TcPOU
FUNCTION_BLOCK FB_PositionX IMPLEMENTS IPosition
VAR_INPUT
END_VAR
VAR_OUTPUT
END_VAR
VAR
	_position	: LREAL;
	_linked		: UDINT;
	_disabled	: BOOL;
	_id	: UDINT;
END_VAR

METHOD Available : BOOL
IF _linked = 0 AND NOT _disabled THEN
	Available := TRUE;
END_IF
END_METHOD

METHOD Disable : BOOL
_disabled := TRUE;
Disable := TRUE;
END_METHOD

METHOD Enable : BOOL
_disabled := FALSE;
Enable := TRUE;
END_METHOD

METHOD GetID : UDINT
GetID := _id;
END_METHOD

METHOD GetPosition : LREAL
GetPosition := _position;
END_METHOD

METHOD SetID : BOOL
VAR_INPUT
	ID	: UDINT;
END_VAR
_id := ID;
END_METHOD

METHOD SetMover : BOOL
VAR_INPUT
	moverNumber	: UDINT;
END_VAR
IF _linked = 0 AND moverNumber <> 0 THEN
	_linked := moverNumber;
	SetMover := TRUE;
END_IF
END_METHOD

METHOD SetPosition
VAR_INPUT
	position	: LREAL;
END_VAR
_position := position;
END_METHOD

END_FUNCTION_BLOCK

// ---- POUs/_NEW/TrackList/FB_Track.TcPOU
FUNCTION_BLOCK FB_Track IMPLEMENTS ITrack
VAR_INPUT
END_VAR
VAR_OUTPUT
END_VAR
VAR
	_list : ARRAY [1..iMaxNumbMovers] OF ST_MoverData;
	_sorted : ARRAY [1..iMaxNumbMovers] OF ST_MoverData;
	_sortedBU : ARRAY [1..iMaxNumbMovers] OF ST_MoverData;
	_tempData : ST_MoverData;
	_temp	: UDINT;
	_mover : ARRAY [1..10] OF IMover;
	i,j : INT;	
END_VAR

METHOD FindMover : UDINT
VAR_INPUT
	status	: INT;
END_VAR
FindMover := 0;
FOR i:= iMaxNumbMovers TO 1 BY -1 DO
	IF _sorted[i].status = status AND NOT _sorted[i].assigned THEN
		_sorted[i].assigned := TRUE;
		FindMover := _sorted[i].id;
		EXIT;
	END_IF
END_FOR
END_METHOD

METHOD SetMoverInUse : BOOL
VAR_INPUT
	moverNumber	: UDINT;
END_VAR
_Sorted[moverNumber].assigned := TRUE;
END_METHOD

METHOD SetMoverRef : BOOL
VAR_INPUT
	index	: DINT;
	mover	: IMover;
END_VAR
_mover[index]:= mover;
END_METHOD

METHOD Sort : BOOL
//backup Cycle Data
_sortedBU := _sorted;

// Step 1: Copy the list
_sorted := _list;

// Step 2: Restore Data
FOR i := 1 TO iMaxNumbMovers DO
	_sorted[i].assigned := _sortedBU[i].assigned;
END_FOR


// Step 2: Bubble Sort the list
FOR i := 1 TO iMaxNumbMovers - 1 DO
    FOR j := i + 1 TO iMaxNumbMovers DO
        IF _sorted[i].pos > _sorted[j].pos THEN
            _tempData := _sorted[i];
            _sorted[i] := _sorted[j];
            _sorted[j] := _tempData;
        END_IF
    END_FOR
END_FOR
END_METHOD

METHOD UpdateMoverData : BOOL
VAR_INPUT
	data	: ST_MoverData;
END_VAR
VAR
	temp	: INT;
END_VAR
_list[data.id] := data;
END_METHOD

END_FUNCTION_BLOCK

// ---- POUs/_NEW/Station/FB_StationX.TcPOU
FUNCTION_BLOCK FB_StationX IMPLEMENTS IStation
VAR_INPUT
END_VAR
VAR_OUTPUT
END_VAR
VAR
	_positions : ARRAY [1..10] OF IPosition;
	_track: ITrack;
	_activePos: IPosition;
	_stateAttract : INT := 1;
	_nextPosition : IPosition;
	_foundMover : UDINT;
	_lastFound : UDINT;
	_size: DINT;
	_i: DINT;
END_VAR

METHOD FindMoverMatch : UDINT
// Find Eligible Mover
IF _activePos <> 0 THEN
	_foundMover := _track.FindMover(status:= _stateAttract);
	IF _foundMover <> 0  AND _foundMover <> _lastFound THEN
		_lastFound := _foundMover;
		_activePos.SetMover(_foundMover);
		_track.SetMoverInUse(_foundMover);		
		//IMover := fbMover[foundMover];
		//IMover.SetPositionID(IPosition.GetID());
	END_IF
END_IF
END_METHOD

METHOD FindNextPosition : IPosition

VAR
	success : BOOL;
END_VAR
// Check sizes
_size := UPPER_BOUND(_positions,1);

// Find First Unassigned Position
_nextPosition := 0;
FOR _i:=1 TO _size DO
	success := _positions[_i].Available();
	IF success THEN
		_nextPosition := _positions[_i];
		EXIT;		
	END_IF
END_FOR

FindNextPosition := _nextPosition;
END_METHOD

METHOD GetMovers : BOOL
THIS^.FindNextPosition();
THIS^.FindMoverMatch();
END_METHOD

METHOD SetPosRef : BOOL
VAR_INPUT
	PosIndex	: DINT;
	PosRef	: REFERENCE TO FB_PositionX;
END_VAR
_positions[PosIndex] := PosRef;
END_METHOD

METHOD SetStationAttraction : BOOL
VAR_INPUT
	setState	: INT;
END_VAR
_stateAttract := setState;
END_METHOD

METHOD SetTrackRef : BOOL
VAR_INPUT
	TrackRef	: ITrack;
END_VAR
_track := TrackRef;
END_METHOD

END_FUNCTION_BLOCK

// ---- POUs/Infeed/Prg_Camming.TcPOU
PROGRAM Prg_Camming
VAR
	bCreateCamTable		: BOOL	:= TRUE;
	CamTable			: MC_CAM_REF;
	MotionFunction 		: ARRAY[1..7] OF MC_MotionFunctionPoint;
	fbCamTable			: MC_CamTableSelect;
	
	rMasterDistance		: LREAL;
	rSlaveDistance		: LREAL;
	rFactor				: LREAL;

END_VAR


CamTable.ArraySize		:= SIZEOF(MotionFunction);
CamTable.NoOfColumns	:= 1;
CamTable.NoOfRows		:= 7;
CamTable.pArray			:= ADR(MotionFunction);
CamTable.TableType		:= MC_TABLETYPE_MOTIONFUNCTION;

rMasterDistance			 	:= GVL_Infeed.rMasterDistance_1Cycle;
rSlaveDistance				:= GVL_Infeed.rDiameterWheel * pi /8;
GVL_Infeed.rSlaveOffset		:= GVL_Infeed.rSyncPosition_Wheel_XTS - (rSlaveDistance * 1.5);
GVL_Infeed.rSlaveOffset_P5 	:= -(GVL_Infeed.rMasterDistance_P5/GVL_Infeed.rMasterDistance_P3)*GVL_Infeed.rSlaveOffset_P3;



// Punt 1
MotionFunction[1].PointIndex		:= 1; 
MotionFunction[1].FunctionType 		:= MOTIONFUNCTYPE_POLYNOM1;
MotionFunction[1].PointType			:= MOTIONPOINTTYPE_MOTION;
MotionFunction[1].RelIndexNextPoint	:= 1;
MotionFunction[1].MasterPos			:= ( 0 * rMasterDistance);
MotionFunction[1].SlavePos			:= ( 0 * rSlaveDistance ) + GVL_Infeed.rSlaveOffset;

// Punt 2
rFactor := ((1.5 * GVL_Infeed.rMasterDistance_1Cycle) - GVL_Infeed.rMasterDistance_P2 )/GVL_Infeed.rMasterDistance_1Cycle;
MotionFunction[2].PointIndex		:= 2; 
MotionFunction[2].FunctionType 		:= MOTIONFUNCTYPE_POLYNOM5_MM;
MotionFunction[2].PointType			:= MOTIONPOINTTYPE_MOTION;
MotionFunction[2].RelIndexNextPoint	:= 1;
MotionFunction[2].MasterPos			:= ( rFactor * rMasterDistance);
MotionFunction[2].SlavePos			:= ( rFactor * rSlaveDistance ) + GVL_Infeed.rSlaveOffset_P2 + GVL_Infeed.rSlaveOffset;

// Punt 3
rFactor := ((1.5 * GVL_Infeed.rMasterDistance_1Cycle) - GVL_Infeed.rMasterDistance_P3 )/GVL_Infeed.rMasterDistance_1Cycle;
MotionFunction[3].PointIndex		:= 3; 
MotionFunction[3].FunctionType 		:= MOTIONFUNCTYPE_POLYNOM1;
MotionFunction[3].PointType			:= MOTIONPOINTTYPE_MOTION;
MotionFunction[3].RelIndexNextPoint	:= 1;
MotionFunction[3].MasterPos			:= ( rFactor * rMasterDistance);
MotionFunction[3].SlavePos			:= ( rFactor * rSlaveDistance ) + GVL_Infeed.rSlaveOffset_P3 + GVL_Infeed.rSlaveOffset;

// Punt 4
MotionFunction[4].PointIndex		:= 4; 
MotionFunction[4].FunctionType 		:= MOTIONFUNCTYPE_POLYNOM1;
MotionFunction[4].PointType			:= MOTIONPOINTTYPE_MOTION;
MotionFunction[4].RelIndexNextPoint	:= 1;
MotionFunction[4].MasterPos			:= ( 1.5 * rMasterDistance);
MotionFunction[4].SlavePos			:= ( 1.5 * rSlaveDistance ) + GVL_Infeed.rSlaveOffset;

// Punt 5
rFactor := ((1.5 * GVL_Infeed.rMasterDistance_1Cycle) + GVL_Infeed.rMasterDistance_P5 )/GVL_Infeed.rMasterDistance_1Cycle;
MotionFunction[5].PointIndex		:= 5; 
MotionFunction[5].FunctionType 		:= MOTIONFUNCTYPE_POLYNOM5_MM;
MotionFunction[5].PointType			:= MOTIONPOINTTYPE_MOTION;
MotionFunction[5].RelIndexNextPoint	:= 1;
MotionFunction[5].MasterPos			:= ( rFactor * rMasterDistance);
MotionFunction[5].SlavePos			:= ( rFactor * rSlaveDistance ) + GVL_Infeed.rSlaveOffset_P5 + GVL_Infeed.rSlaveOffset;

// Punt 6
rFactor := ((1.5 * GVL_Infeed.rMasterDistance_1Cycle) + GVL_Infeed.rMasterDistance_P6 )/GVL_Infeed.rMasterDistance_1Cycle;
MotionFunction[6].PointIndex		:= 6; 
MotionFunction[6].FunctionType 		:= MOTIONFUNCTYPE_POLYNOM1;
MotionFunction[6].PointType			:= MOTIONPOINTTYPE_MOTION;
MotionFunction[6].RelIndexNextPoint	:= 0;
MotionFunction[6].MasterPos			:= ( rFactor * rMasterDistance);
MotionFunction[6].SlavePos			:= ( rFactor * rSlaveDistance ) + GVL_Infeed.rSlaveOffset;

// Punt 7
MotionFunction[7].PointIndex		:= 7; 
MotionFunction[7].PointType			:= MOTIONPOINTTYPE_MOTION;
MotionFunction[7].RelIndexNextPoint	:= 0;
MotionFunction[7].MasterPos			:= ( 3 * rMasterDistance);
MotionFunction[7].SlavePos			:= ( 3 * rSlaveDistance ) + GVL_Infeed.rSlaveOffset;

// Create Cam Table
fbCamTable(
	Master		:= GVL_Infeed.MasterAxis, 
	Slave		:= GVL_Infeed.VirtalMaster[1], 
	CamTable	:= CamTable, 
	Execute		:= bCreateCamTable, 
	Periodic	:= TRUE, 
	CamTableID	:= 1, 
	);

END_PROGRAM
